{attribute addProperty BoxType "EJ1914-0000-0017"}
{attribute addProperty Id "FSoE_CommandUSINT811FSIN_Module_1_Channel_1_InputBIT10.1251FSIN_Module_1_Channel_2_InputBIT10.1252FSIN_Module_1_Module_FaultBIT10.1251FSIN_Module_2_Channel_1_InputBIT10.1251FSIN_Module_2_Channel_2_InputBIT10.1252FSIN_Module_2_Module_FaultBIT10.1251FSoE_CRC_000UINT1623FSoE_Connection_IDUINT1622"}
{attribute addProperty CRC "1263750294"}
{attribute addProperty SizeInBites "48"}
{attribute addProperty SizeInBytes "6"}
TYPE FSOE_4B534C96 :
STRUCT
	{attribute addProperty Name "FSoE_Command"}
	FSoE_Command : USINT;
	{attribute addProperty Name "FSIN_Module_1_Channel_1_Input"}
	FSIN_Module_1_Channel_1_Input : BOOL;
	{attribute addProperty Name "FSIN_Module_1_Channel_2_Input"}
	FSIN_Module_1_Channel_2_Input : BOOL;
	{attribute addProperty Name "FSIN_Module_1_Module_Fault"}
	FSIN_Module_1_Module_Fault : BOOL;
	{attribute addProperty Name "FSIN_Module_2_Channel_1_Input"}
	FSIN_Module_2_Channel_1_Input : BOOL;
	{attribute addProperty Name "FSIN_Module_2_Channel_2_Input"}
	FSIN_Module_2_Channel_2_Input : BOOL;
	{attribute addProperty Name "FSIN_Module_2_Module_Fault"}
	FSIN_Module_2_Module_Fault : BOOL;
	{attribute 'hide'}
	reserve_1_BIT_0 : BOOL;
	{attribute 'hide'}
	reserve_1_BIT_1 : BOOL;
	{attribute addProperty Name "FSoE_CRC_000"}
	FSoE_CRC_000 : UINT;
	{attribute addProperty Name "FSoE_Connection_ID"}
	FSoE_Connection_ID : UINT;
END_STRUCT
END_TYPE

(* stored: Version 1.2.0.0, ProductVersion 3.1.4024.9
   DUT FSOE_4B534C96: Id {53cb1134-a3fd-4786-ad28-f4a17762fb4a} *)
